{region '#Template'}
	{attribute 'Version' := '5.0.0.0'}
	{attribute 'Tags' := '"LCID": "1031", "Text": "Universal, Analog, Aggregate"'}
	{attribute 'Tags' := '"LCID": "1033", "Text": "Universal, Analog, Aggregate"'}
	{attribute 'Using' := '"Type": "Template", "URI": "EC_ID"'}
	{attribute 'Using' := '"Type": "Template", "URI": "BA2_Param"'}
	{attribute 'Description' := '"LCID": "1031", "Text": "Aktor binär"'}
	{attribute 'Description' := '"LCID": "1033", "Text": "Actuator binary"'}
{endregion}
FUNCTION_BLOCK FB_BA_ActuatorCmd EXTENDS FB_BA_View
VAR_INPUT
	stCmd						: ST_BA_Binary;	
END_VAR
VAR_OUTPUT
	bCmd						: BOOL;
	bDst						: BOOL;
	eActivePrio					: E_BA_Priority;
END_VAR
VAR_INPUT CONSTANT
	Cmd							: FB_BA_BO_Raw;		
	PlantLock					: FB_BA_PlantLock;								
END_VAR
VAR
	bPrioSfty					: BOOL;
	bPrioCrit					: BOOL;	
END_VAR
VAR // added by the converter: edge detectors and wires of the graphical bodies
    _w1 : ANY;
END_VAR

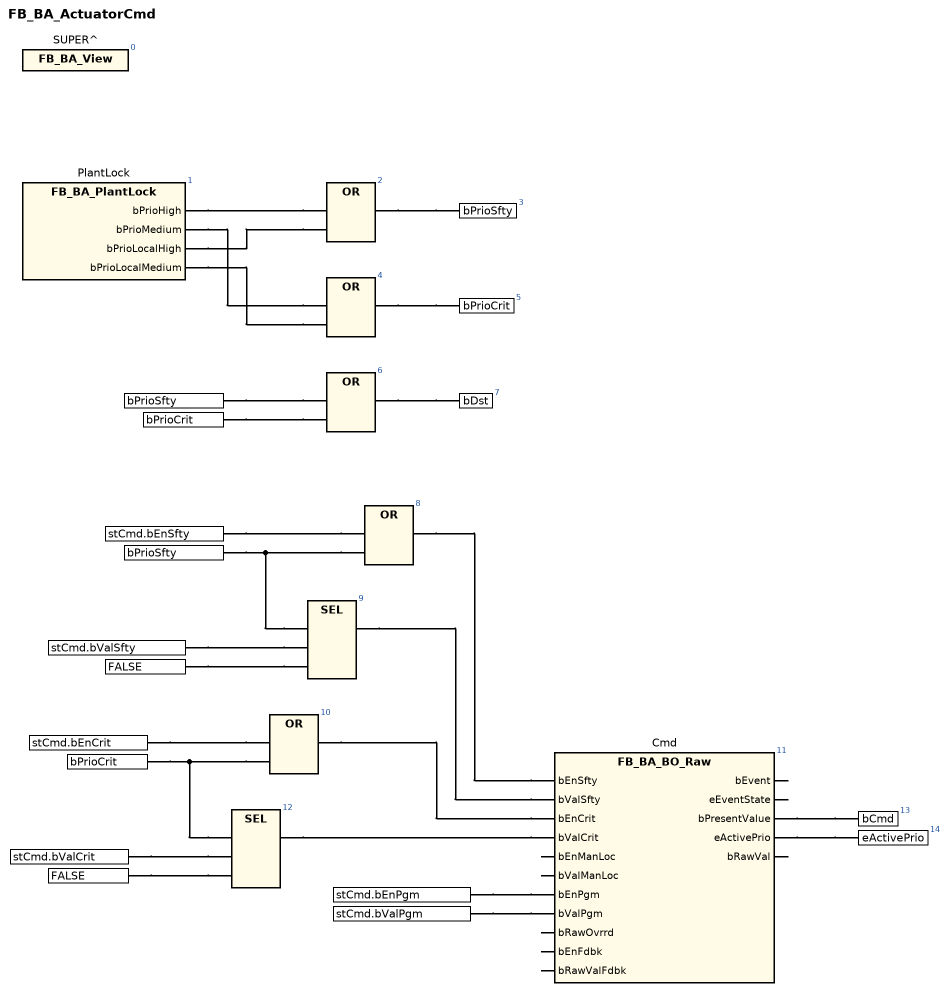
SUPER^(); // FB_BA_View
PlantLock(); // FB_BA_PlantLock
bPrioSfty := PlantLock.bPrioHigh OR PlantLock.bPrioLocalHigh;
bPrioCrit := PlantLock.bPrioMedium OR PlantLock.bPrioLocalMedium;
bDst := bPrioSfty OR bPrioCrit;
Cmd(
    bEnSfty := stCmd.bEnSfty OR bPrioSfty,
    bValSfty := SEL(bPrioSfty, stCmd.bValSfty, FALSE),
    bEnCrit := stCmd.bEnCrit OR bPrioCrit,
    bValCrit := _w1,
    bEnPgm := stCmd.bEnPgm,
    bValPgm := stCmd.bValPgm); // FB_BA_BO_Raw
_w1 := SEL(bPrioCrit, stCmd.bValCrit, FALSE);
bCmd := Cmd.bPresentValue;
eActivePrio := Cmd.eActivePrio;

METHOD FB_init : BOOL
VAR_INPUT
	bInitRetains : BOOL; // if TRUE, the retain variables are initialized (warm start / cold start)
	bInCopyCode : BOOL;  // if TRUE, the instance afterwards gets moved into the copy code (online change)
END_VAR
PlantLock.Parent					:= THIS^;		

Cmd.iParent							:= THIS^;
Cmd.iLabel							:= LblFun_SwitchingCommand;  
Cmd.ePolarity						:= E_BA_Polarity.eNormal;
Cmd.sActiveText 					:= txtEvent_On;
Cmd.sInactiveText 					:= txtEvent_Off;
Cmd.bEnManualRm						:= FALSE;	//	Priority  8	
Cmd.bValManualRm					:= FALSE;	//	Priority  8
Cmd.nEventClassID					:= EC_ID.NC40;
Cmd.stTimeDelay.nToNormal			:= BA2_Param.nDefTimeDelay_ToNormal;
Cmd.stTimeDelay.nToAbnormal			:= BA2_Param.nDefTimeDelay_ToAbnormal;
Cmd.aEventTransitionText[1]			:= txtEvent_Disturb;
Cmd.aEventTransitionText[2]			:= txtEvent_None;
Cmd.aEventTransitionText[3]			:= txtEvent_Normal;
Cmd.bEventDetectionEnable			:= FALSE;
Cmd.eEnPlantLock					:= E_BA_LockPriority.eNoLock;
END_METHOD

END_FUNCTION_BLOCK

(* stored: Version 1.1.0.1, ProductVersion 3.1.4024.12
   POU FB_BA_ActuatorCmd: Id {d324037e-60db-4717-9d08-593d44dbd1e2}, SpecialFunc None
   Method FB_init: Id {b90a9b9f-7987-4590-908b-29b6ee3fc5aa} *)
